Staubli VAL3: staubli.dtx

jointRx a[5]
  [0] = {j1=-30.841182, j2=5.759125, j3=4.776611, j4=-4.337769, j5=0.185181, j6=-0.440956}
  [1] = {j1=85.144596, j2=41.264374, j3=85.057123, j4=50.225892, j5=66.231894, j6=10.998627}
  [2] = {j1=68.499734, j2=-4.868335, j3=97.031411, j4=43.922331, j5=74.239113, j6=-0.440956}
  [3] = {j1=68.499734, j2=-4.868335, j3=97.031411, j4=-108.057669, j5=-94.510887, j6=-0.440956}
  [4] = {j1=71.019734, j2=14.816197, j3=97.031411, j4=-108.057669, j5=-94.510887, j6=-0.440956}
mdesc vit
mdesc vitesse = {accel=1}
num i = 5
pointRx s = {x=-8.69, y=271.759218, z=117.046845, rx=-153.130649, ry=-73.218542, rz=-38.514559, fatherId=world[0]}
pointRx w = {x=-8.691937, y=354.195721, z=-66.105143, rx=-153.13277, ry=-73.21809, rz=-38.515963, fatherId=world[0]}
